(* PLC project Tc2_Utilities.PULARGE_TO_ULARGE Demo, tc3-libraries-kb TwinCAT 3.1 *)
(* stored: creationDateTime 2026-05-10T15:00:00, modificationDateTime 2026-05-10T15:00:00 *)

PROGRAM P_Demo_PULARGE_TO_ULARGE
  VAR
    rResult : T_ULARGE_INTEGER;  (* PULARGE_TO_ULARGE 返回值 *)
    bRun : BOOL;  (* 触发一次调用 *)
    v : T_ULARGE_INTEGER;  (* 测试用本地变量（取址） *)
  END_VAR

            // ============================================================
// Tc2_Utilities.PULARGE_TO_ULARGE 演示程序（FUNCTION）
// ============================================================
// 验证步骤：
//   1. 引用 Tc2_Utilities
//   2. 编译 + 登录
//   3. 强制 bRun := TRUE 一个周期
//   4. 在线监视 rResult 应等于 v 的当前值
// ============================================================

IF bRun THEN
    rResult := PULARGE_TO_ULARGE(ADR(v));
    bRun := FALSE;
END_IF;

          
END_PROGRAM
